# EPICS StreamDevice protocol: protocols/v2f.proto
Terminator = LF;
ExtraInput = Ignore;
ReplyTimeout = 2500;

setFreqFun {
	out "v2f_freq_\$1_\$2 %d";
}

setHF {
	out "hf %d";
}

setSrcMap {
	out "chan_sel %(A)d,%(B)d,%(C)d,%(D)d";
}
